// TIA Portal V19 export
FUNCTION_BLOCK "LiftSeq"   // FB12, GRAPH
TITLE = LiftSeq
AUTHOR : Siemens
// Graph sequence BeltLift
// stored: GraphVersion 6.0, InitialValuesAcquisition true, IsIECCheckEnabled true, LanguageInNetworks FBD, SetENOAutomatically true
   // inherited from GRAPH_BASE
   VAR_INPUT
      OFF_SQ { ExternalWritable := 'False'} : Bool := false;   // Kette ausschalten / Turn sequence off
      INIT_SQ { ExternalWritable := 'False'} : Bool := false;   // Kette in Initialzustand versetzen / Set sequence to initial state
      ACK_EF { ExternalWritable := 'False'} : Bool := false;   // Alle Fehler und Störungen quittieren / Acknowledge all errors and faults
      REG_EF { ExternalWritable := 'False'} : Bool := false;   // Register all errors and faults / Alle Fehler und Störungen registrieren
      ACK_S { ExternalWritable := 'False'} : Bool := false;   // Acknowledge step indicated in S_NO / Schritt quittieren, der an Parameter S_NO anliegt
      REG_S { ExternalWritable := 'False'} : Bool := false;   // Register the step indicated in S_NO / Schritt registrieren, der an Parameter S_NO anliegt
      HALT_SQ { ExternalWritable := 'False'} : Bool := false;   // Halt sequence immediately / Kette sofort anhalten
      HALT_TM { ExternalWritable := 'False'} : Bool := false;   // Halt timers immediately / Zeiten sofort anhalten
      ZERO_OP { ExternalWritable := 'False'} : Bool := false;   // Set all operands assigned with N, L, D to 0 / Alle mit N, L, D zugewiesenen Operanden auf 0 setzen
      EN_IL { ExternalWritable := 'False'} : Bool := false;   // Activate interlocks / Interlockbearbeitung aktivieren
      EN_SV { ExternalWritable := 'False'} : Bool := false;   // Activate supervision processing / Supervisionsbearbeitung aktivieren
      EN_ACKREQ { ExternalWritable := 'False'} : Bool := false;   // Activate mandatory acknowledgment / Quittierpflicht aktivieren
      EN_SSKIP { ExternalWritable := 'False'} : Bool := false;   // Enable "Skip step" / "Schritte überspringen" aktivieren
      DISP_SACT { ExternalWritable := 'False'} : Bool := false;   // Display active steps only / Nur aktive Schritte anzeigen
      DISP_SEF { ExternalWritable := 'False'} : Bool := false;   // Display only steps with errors and disrupted steps / Nur fehlerhafte und gestörte Schritte anzeigen
      DISP_SALL { ExternalWritable := 'False'} : Bool := false;   // Display all steps / Alle Schritte anzeigen
      S_PREV { ExternalWritable := 'False'} : Bool := false;   // Vorherigen Schritt am Parameter S_NO ausgeben / Output previous step in parameter S_NO
      S_NEXT { ExternalWritable := 'False'} : Bool := false;   // Nächsten Schritt am Parameter S_NO anzeigen / Indicate next step in parameter S_NO
      SW_AUTO { ExternalWritable := 'False'} : Bool := false;   // Automtischer Betrieb / Automatic mode
      SW_TAP { ExternalWritable := 'False'} : Bool := false;   // Halbautomatisch/Weiterschalten mit Transition / Semiautomatic/switch with transition
      SW_TOP { ExternalWritable := 'False'} : Bool := false;   // Halbautomatisch/Ignoriere Transition / Semiautomatic/ignore transition
      SW_MAN { ExternalWritable := 'False'} : Bool := false;   // Handbetrieb / Manual mode
      S_SEL { ExternalWritable := 'False'} : Int := 0;   // Schritt auswählen, der an S_NO ausgegeben werden soll / Select step to be output to S_NO
      S_SELOK { ExternalWritable := 'False'} : Bool := false;   // Enter value from S_SEL in S_NO / Wert aus S_SEL nach S_NO übernehmen
      S_ON { ExternalWritable := 'False'} : Bool := false;   // Schritt aktivieren, der an Parameter S_NO anliegt / Activate step indicated in S_NO
      S_OFF { ExternalWritable := 'False'} : Bool := false;   // Schritt deaktivieren, der an Parameter S_NO anliegt / Deactivate step indicated S_NO
      T_PREV { ExternalWritable := 'False'} : Bool := false;   // Display previous transition in T_NO / Vorherige Transition an Parameter T_NO anzeigen
      T_NEXT { ExternalWritable := 'False'} : Bool := false;   // Display next transition at parameter T_NO / Nächste Transition an Parameter T_NO anzeigen
      T_PUSH { ExternalWritable := 'False'} : Bool := false;   // Schaltfreigabe für Transition im halbautomatischen Betrieb / Enable transition to switch in semi automatic mode
      EN_LMODE { ExternalWritable := 'False'} : Bool := false;   // Activate learning mode / Lernmodus aktivieren
      RESET_CRIT { ExternalWritable := 'False'} : Bool := false;   // Reset all initial values recorded for interlocks and transitions / Alle Erstwerte, die für Interlocks und Transitionen aufgezeichnet wurden, zurücksetzen
   END_VAR
   VAR_OUTPUT
      S_NO { ExternalWritable := 'False'} : Int := 0;   // Schrittnummer / Step number
      S_MORE { ExternalWritable := 'False'} : Bool := false;   // Weitere Schritte sind vorhanden und können in S_NO angezeigt werden. / More steps are available and can be shown in S_NO
      S_ACTIVE { ExternalWritable := 'False'} : Bool := false;   // Schritt, der an Parameter S_NO angezeigt wird, ist aktiv / Step indicated in S_NO is active
      S_TIME { ExternalWritable := 'False'} : Time := T#0ms;   // Step activation time / Schrittaktivierungszeit
      S_TIMEOK { ExternalWritable := 'False'} : Time := T#0ms;   // No error in step activation time / Schrittaktivierungszeit fehlerfrei
      S_CRITLOC { ExternalWritable := 'False'} : DWord := 16#0;   // Interlock criteria bits / Interlock-Kriterienbits
      S_CRITLOCERR { ExternalWritable := 'False'} : DWord := 16#0;   // Interlock criteria bits for event L1 / Interlock-Kriterienbits bei Ereignis L1
      S_STATE { ExternalWritable := 'False'} : Word := 16#0;   // Step state bits / Schrittzustandsbits
      T_NO { ExternalWritable := 'False'} : Int := 0;   // Transition number / Transitionsnummer
      T_MORE { ExternalWritable := 'False'} : Bool := false;   // More valid transitions available for display / Weitere gültige Transitionen zur Anzeige verfügbar
      T_CRIT { ExternalWritable := 'False'} : DWord := 16#0;   // Transition criteria bits / Transitions-Kriterienbits
      T_CRITOLD { ExternalWritable := 'False'} : DWord := 16#0;   // Transition criteria bits from last cycle / Transitions-Kriterienbits des letzten Zyklus
      T_CRITFLT { ExternalWritable := 'False'} : DWord := 16#0;   // Transition criteria bits for event V1 / Transitions-Kriterienbits bei Ereignis V1
      ERROR { ExternalWritable := 'False'} : Bool := false;   // Interlock group error / Sammelfehler Interlock
      FAULT { ExternalWritable := 'False'} : Bool := false;   // Supervision group error / Sammelfehler Supervision
      ERR_FLT { ExternalWritable := 'False'} : Bool := false;   // Sammelfehler Interlock oder Supervision / Interlock or supervision group error
      SQ_ISOFF { ExternalWritable := 'False'} : Bool := false;   // Sequence is off (no step active) / Kette ausgeschaltet (kein Schritt aktiv)
      SQ_HALTED { ExternalWritable := 'False'} : Bool := false;   // Sequence halted / Kette angehalten
      TM_HALTED { ExternalWritable := 'False'} : Bool := false;   // Timers halted / Zeiten angehalten
      OP_ZEROED { ExternalWritable := 'False'} : Bool := false;   // All the operands assigned with N, L, D are set to 0 / Alle mit N, L oder D zugewiesenen Operanden auf 0 gesetzt
      IL_ENABLED { ExternalWritable := 'False'} : Bool := false;   // Interlocks are active / Interlockbearbeitung aktiv
      SV_ENABLED { ExternalWritable := 'False'} : Bool := false;   // Supervision processing activated / Supervisionsbearbeitung aktiviert
      ACKREQ_ENABLED { ExternalWritable := 'False'} : Bool := false;   // Mandatory acknowledgment activated / Quittierpflicht aktiviert
      SSKIP_ENABLED { ExternalWritable := 'False'} : Bool := false;   // Skip steps activated / Schritte überspringen aktiviert
      SACT_DISP { ExternalWritable := 'False'} : Bool := false;   // Display active steps only / Nur aktive Schritte anzeigen
      SEF_DISP { ExternalWritable := 'False'} : Bool := false;   // Display only steps with errors or disrupted steps / Nur fehlerhafte oder gestörte Schritte anzeigen
      SALL_DISP { ExternalWritable := 'False'} : Bool := false;   // Display all steps / Alle Schritte anzeigen
      AUTO_ON { ExternalWritable := 'False'} : Bool := false;   // Automatischer Betrieb eingeschaltet / Automatic mode is active
      TAP_ON { ExternalWritable := 'False'} : Bool := false;   // Halbautomatischer Betrieb/Schritt mit Transition eingeschaltet / Semiautomatic mode/step with transition enabled
      TOP_ON { ExternalWritable := 'False'} : Bool := false;   // Halbautomatischer Betrieb/Ignoriere Transition eingeschaltet / Semiautomatic mode/ignore transition enabled
      MAN_ON { ExternalWritable := 'False'} : Bool := false;   // Handbetrieb eingeschaltet / Manual mode is active
      LMODE_ENABLED { ExternalWritable := 'False'} : Bool := false;   // Learning mode is active / Lernmodus aktiv
   END_VAR
BEGIN
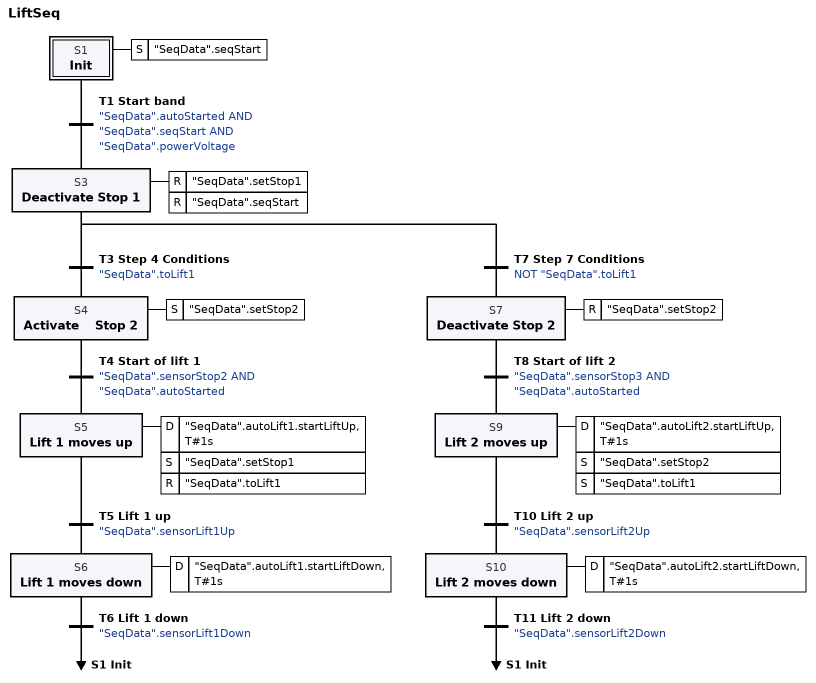
   // sequencer 1
   INITIAL_STEP Init:   // S1, max time T#10S, warning time T#7S
              S    "SeqData".seqStart
   END_STEP
   TRANSITION "Start band" FROM Init TO "Deactivate Stop 1"   // T1
      := "SeqData".autoStarted AND "SeqData".seqStart AND "SeqData".powerVoltage;
   END_TRANSITION
   STEP "Deactivate Stop 1":   // S3, max time T#10S, warning time T#7S
              R    "SeqData".setStop1
              R    "SeqData".seqStart
   END_STEP
   TRANSITION "Step 4 Conditions" FROM "Deactivate Stop 1" TO "Activate    Stop 2"   // T3
      := "SeqData".toLift1;
   END_TRANSITION
   TRANSITION "Step 7 Conditions" FROM "Deactivate Stop 1" TO "Deactivate Stop 2"   // T7
      := NOT "SeqData".toLift1;
   END_TRANSITION
   STEP "Activate    Stop 2":   // S4, max time T#10S, warning time T#7S
              S    "SeqData".setStop2
   END_STEP
   TRANSITION "Start of lift 1" FROM "Activate    Stop 2" TO "Lift 1 moves up"   // T4
      := "SeqData".sensorStop2 AND "SeqData".autoStarted;
   END_TRANSITION
   STEP "Lift 1 moves up":   // S5, max time T#10S, warning time T#7S
      interlock C := "SeqData".doorClosed AND "SeqData".liftFree;   // Door at lift not closed or lift blocked. / Tür an Hubeinheit nicht geschlossen oder Hubeinheit blockiert.
      supervision V := #"Lift 1 moves up".T > T#5S;   // Lift1 upper position not reached / Hubeinheit 1obere Position nicht erreicht
              D    "SeqData".autoLift1.startLiftUp, T#1s
              S    "SeqData".setStop1
              R    "SeqData".toLift1
   END_STEP
   TRANSITION "Lift 1 up" FROM "Lift 1 moves up" TO "Lift 1 moves down"   // T5
      := "SeqData".sensorLift1Up;
   END_TRANSITION
   STEP "Lift 1 moves down":   // S6, max time T#10S, warning time T#7S
      interlock C := "SeqData".doorClosed AND "SeqData".liftFree;   // Door at lift not closed or lift blocked. / Tür an Hubeinheit nicht geschlossen oder Hubeinheit blockiert.
      supervision V := #"Lift 1 moves down".T > T#5S;   // Lift1 lower position not reached / Hubeinheit 1 untere Position nicht erreicht
              D    "SeqData".autoLift1.startLiftDown, T#1s
   END_STEP
   TRANSITION "Lift 1 down" FROM "Lift 1 moves down" TO Init   // T6, jump
      := "SeqData".sensorLift1Down;
   END_TRANSITION
   STEP "Deactivate Stop 2":   // S7, max time T#10S, warning time T#7S
              R    "SeqData".setStop2
   END_STEP
   TRANSITION "Start of lift 2" FROM "Deactivate Stop 2" TO "Lift 2 moves up"   // T8
      := "SeqData".sensorStop3 AND "SeqData".autoStarted;
   END_TRANSITION
   STEP "Lift 2 moves up":   // S9, max time T#10S, warning time T#7S
      interlock C := "SeqData".doorClosed AND "SeqData".liftFree;   // Door at lift not closed or lift blocked. / Tür an Hubeinheit nicht geschlossen oder Hubeinheit blockiert.
      supervision V := #"Lift 2 moves up".T > T#5S;   // Lift2 upper position not reached / Hubeinheit 2 obere Position nicht erreicht
              D    "SeqData".autoLift2.startLiftUp, T#1s
              S    "SeqData".setStop2
              S    "SeqData".toLift1
   END_STEP
   TRANSITION "Lift 2 up" FROM "Lift 2 moves up" TO "Lift 2 moves down"   // T10
      := "SeqData".sensorLift2Up;
   END_TRANSITION
   STEP "Lift 2 moves down":   // S10, max time T#10S, warning time T#7S
      interlock C := "SeqData".doorClosed AND "SeqData".liftFree;   // Door at lift not closed or lift blocked. / Tür an Hubeinheit nicht geschlossen oder Hubeinheit blockiert.
      supervision V := #"Lift 2 moves down".T > T#5S;   // Lift2 lower position not reached / Hubeinheit 2 untere Position nicht erreicht
              D    "SeqData".autoLift2.startLiftDown, T#1s
   END_STEP
   TRANSITION "Lift 2 down" FROM "Lift 2 moves down" TO Init   // T11, jump
      := "SeqData".sensorLift2Down;
   END_TRANSITION
END_FUNCTION_BLOCK
